//////////////轴位置赋初值////////////
IF arrAxisPar[AxisNo.BuffeLine].arrTargetPoint[1]=0 THEN
	arrAxisPar[AxisNo.BuffeLine].arrTargetPoint[1]:=20;
END_IF
IF arrAxisPar[AxisNo.Mould].arrTargetPoint[1]=0 THEN
	arrAxisPar[AxisNo.Mould].arrTargetPoint[1]:=230;
END_IF
IF arrAxisPar[AxisNo.Mould].arrTargetPoint[2]=0 THEN
	arrAxisPar[AxisNo.Mould].arrTargetPoint[2]:=130;
END_IF
IF arrAxisPar[AxisNo.Cuter].arrTargetPoint[1]=0 THEN
	arrAxisPar[AxisNo.Cuter].arrTargetPoint[1]:=230;
END_IF
IF arrAxisPar[AxisNo.Cuter].arrTargetPoint[2]=0 THEN
	arrAxisPar[AxisNo.Cuter].arrTargetPoint[2]:=130;
END_IF
IF arrAxisPar[AxisNo.CCDPressPush].arrTargetPoint[1]=0 THEN
	arrAxisPar[AxisNo.CCDPressPush].arrTargetPoint[1]:=200;
END_IF
IF arrAxisPar[AxisNo.CCDPressPush].arrTargetPoint[2]=0 THEN
	arrAxisPar[AxisNo.CCDPressPush].arrTargetPoint[2]:=180;
END_IF
(*
IF arrAxisPar[AxisNo.NGPush1].arrTargetPoint[1]=0 THEN
	arrAxisPar[AxisNo.NGPush1].arrTargetPoint[1]:=1;
END_IF
IF arrAxisPar[AxisNo.NGPush1].arrTargetPoint[2]=0 THEN
	arrAxisPar[AxisNo.NGPush1].arrTargetPoint[2]:=180;
END_IF
IF arrAxisPar[AxisNo.NGPush2].arrTargetPoint[1]=0 THEN
	arrAxisPar[AxisNo.NGPush2].arrTargetPoint[1]:=270;
END_IF
IF arrAxisPar[AxisNo.NGPush2].arrTargetPoint[2]=0 THEN
	arrAxisPar[AxisNo.NGPush2].arrTargetPoint[2]:=90;
END_IF
*)
IF arrAxisPar[AxisNo.MouldRectify_X].arrTargetPoint[1]=0 THEN
	arrAxisPar[AxisNo.MouldRectify_X].arrTargetPoint[1]:=1;
END_IF
IF arrAxisPar[AxisNo.MouldRectify_X].arrTargetPoint[2]=0 THEN
	arrAxisPar[AxisNo.MouldRectify_X].arrTargetPoint[2]:=2;
END_IF
IF arrAxisPar[AxisNo.MouldRectify_Y].arrTargetPoint[1]=0 THEN
	arrAxisPar[AxisNo.MouldRectify_Y].arrTargetPoint[1]:=1;
END_IF
IF arrAxisPar[AxisNo.MouldRectify_Y].arrTargetPoint[2]=0 THEN
	arrAxisPar[AxisNo.MouldRectify_Y].arrTargetPoint[2]:=2;
END_IF
IF arrAxisPar[AxisNo.CuterBeltChange].arrTargetPoint[1]=0 THEN
	arrAxisPar[AxisNo.CuterBeltChange].arrTargetPoint[1]:=1;
END_IF
IF arrAxisPar[AxisNo.CuterBeltChange].arrTargetPoint[2]=0 THEN
	arrAxisPar[AxisNo.CuterBeltChange].arrTargetPoint[2]:=2;
END_IF
IF arrAxisPar[AxisNo.CuterDegRectify].arrTargetPoint[1]=0 THEN
	arrAxisPar[AxisNo.CuterDegRectify].arrTargetPoint[1]:=0.1;
END_IF
IF arrAxisPar[AxisNo.CuterDegRectify].arrTargetPoint[2]=0 THEN
	arrAxisPar[AxisNo.CuterDegRectify].arrTargetPoint[2]:=0.2;
END_IF
//监控极耳数据
TabData[1].fPhotoPosC;TabData[1].fPhotoPosM;TabData[1].fTab_OffsetC;TabData[1].fTab_OffsetM;
TabData[2].fPhotoPosC;TabData[2].fPhotoPosM;TabData[2].fTab_OffsetC;TabData[2].fTab_OffsetM;
TabData[3].fPhotoPosC;TabData[3].fPhotoPosM;TabData[3].fTab_OffsetC;TabData[3].fTab_OffsetM;
TabData[4].fPhotoPosC;TabData[4].fPhotoPosM;TabData[3].fTab_OffsetC;TabData[4].fTab_OffsetM;
TabData[5].fPhotoPosC;TabData[5].fPhotoPosM;TabData[5].fTab_OffsetC;TabData[5].fTab_OffsetM;
TabData[6].fPhotoPosC;TabData[6].fPhotoPosM;TabData[6].fTab_OffsetC;TabData[6].fTab_OffsetM;
TabData[7].fPhotoPosC;TabData[7].fPhotoPosM;TabData[7].fTab_OffsetC;TabData[7].fTab_OffsetM;
TabData[8].fPhotoPosC;TabData[8].fPhotoPosM;TabData[8].fTab_OffsetC;TabData[8].fTab_OffsetM;
TabData[9].fPhotoPosC;TabData[9].fPhotoPosM;TabData[9].fTab_OffsetC;TabData[9].fTab_OffsetM;
TabData[10].fPhotoPosC;TabData[10].fPhotoPosM;TabData[10].fTab_OffsetC;TabData[10].fTab_OffsetM;
//监控极耳间距数据
InteData[1].fTabIntervalC;InteData[1].fTabIntervalM;InteData[1].bLineScanNG;
InteData[2].fTabIntervalC;InteData[2].fTabIntervalM;InteData[2].bLineScanNG;
InteData[3].fTabIntervalC;InteData[3].fTabIntervalM;InteData[3].bLineScanNG;
InteData[4].fTabIntervalC;InteData[4].fTabIntervalM;InteData[4].bLineScanNG;
InteData[5].fTabIntervalC;InteData[5].fTabIntervalM;InteData[5].bLineScanNG;
InteData[6].fTabIntervalC;InteData[6].fTabIntervalM;InteData[6].bLineScanNG;
InteData[7].fTabIntervalC;InteData[7].fTabIntervalM;InteData[7].bLineScanNG;
InteData[8].fTabIntervalC;InteData[8].fTabIntervalM;InteData[8].bLineScanNG;
InteData[9].fTabIntervalC;InteData[9].fTabIntervalM;InteData[9].bLineScanNG;
InteData[10].fTabIntervalC;InteData[10].fTabIntervalM;InteData[10].bLineScanNG;

IF bTest[1] THEN
	arrAxisCtrl[VirAxisNo.VirMain].Cmd.bDynamitcsParSel:=1;
	arrAxisCtrl[VirAxisNo.VirMain].Cmd.fPositon_of_Abs:=arrAxisCtrl[VirAxisNo.VirMain].Status.fActPos-arrAxisCtrl[VirAxisNo.VirMain].Status.fModuloActPos+720;
	//arrAxisPar[VirAxisNo.VirMain].fTagatTime:=((arrAxisCtrl[VirAxisNo.VirMain].Cmd.fPositon_of_Abs-arrAxisCtrl[VirAxisNo.VirMain].Status.fActPos)/360) *60/PolePar.iMainVel+0.05 ;
	arrAxisPar[VirAxisNo.VirMain].fVelocity_of_Abs:=PolePar.iMainVel*6;
	arrAxisCtrl[VirAxisNo.VirMain].Cmd.bMoveAbs:=TRUE;
	bTest[1]:=FALSE;
END_IF

ftest1:=FC_LengthToAngle(CCD_COM.fDemLength,PolePar.Machine.fMQDriverDiameter);
(*
arrAxisCtrl[VirAxisNo.VirMain].Status.Moving;     arrAxisCtrl[VirAxisNo.VirMain].Status.fActPos;
IF bTest[2] THEN
	arrAxisCtrl[VirAxisNo.VirMain].Cmd.bDynamitcsParSel:=1;
	ftest2:=arrAxisCtrl[VirAxisNo.VirMain].Status.fActPos+360;
	arrAxisCtrl[VirAxisNo.VirMain].Cmd.fPositon_of_Abs:=ftest2;
	//arrAxisPar[VirAxisNo.VirMain].fTagatTime:=((arrAxisCtrl[VirAxisNo.VirMain].Cmd.fPositon_of_Abs-arrAxisCtrl[VirAxisNo.VirMain].Status.fActPos)/360) *60/PolePar.iMainVel+0.05 ;
	arrAxisPar[VirAxisNo.VirMain].fVelocity_of_Abs:=20;
	arrAxisCtrl[VirAxisNo.VirMain].Cmd.bMoveAbs:=TRUE;
	itest:=2;
bTest[2]:=FALSE;
END_IF
IF bTest[3] THEN
	arrAxisCtrl[VirAxisNo.VirMain].Cmd.bDynamitcsParSel:=1;
	ftest3:=arrAxisCtrl[VirAxisNo.VirMain].Status.fActPos-arrAxisCtrl[VirAxisNo.VirMain].Status.fModuloActPos+720;
	arrAxisCtrl[VirAxisNo.VirMain].Cmd.fPositon_of_Abs:=ftest3;
	//arrAxisPar[VirAxisNo.VirMain].fTagatTime:=((arrAxisCtrl[VirAxisNo.VirMain].Cmd.fPositon_of_Abs-arrAxisCtrl[VirAxisNo.VirMain].Status.fActPos)/360) *60/PolePar.iMainVel+0.05 ;
	arrAxisPar[VirAxisNo.VirMain].fVelocity_of_Abs:=20;
	arrAxisCtrl[VirAxisNo.VirMain].Cmd.bMoveAbs:=TRUE;
	itest:=3;
bTest[3]:=FALSE;
END_IF
*)
IF btest[2] THEN
	MEMSET(ADR(fM_TabInterData),0,SIZEOF(fM_TabInterData)); //  
	btest[2]:=FALSE;
END_IF
IF btest[3] THEN
	MEMSET(ADR(fDriverOffsetData),0,SIZEOF(fDriverOffsetData)); //  
	btest[3]:=FALSE;
END_IF
IF btest[4] THEN
	//MEMSET(ADR(),0,SIZEOF()); //  
	btest[4]:=FALSE;
END_IF
IF btest[5] THEN
	//MEMSET(ADR(),0,SIZEOF()); //  
	btest[5]:=FALSE;
	fDegreeRec1:=FC_Variance(fOffsetDeg);		
END_IF



(*
IF NOT InterPart.M1Safety THEN
   arrAxisCtrl[AxisNo.SubBelt1].Cmd.JogP_Condition:=TRUE;
   arrAxisCtrl[AxisNo.SubBelt1].Cmd.JogN_Condition:=TRUE;
ELSE 
   arrAxisCtrl[AxisNo.SubBelt1].Cmd.JogP_Condition:=FALSE;
   arrAxisCtrl[AxisNo.SubBelt1].Cmd.JogN_Condition:=FALSE;
END_IF

IF NOT InterPart.M2Safety THEN
   arrAxisCtrl[AxisNo.SubBelt2].Cmd.JogP_Condition:=TRUE;
   arrAxisCtrl[AxisNo.SubBelt2].Cmd.JogN_Condition:=TRUE;
ELSE 
   arrAxisCtrl[AxisNo.SubBelt2].Cmd.JogP_Condition:=FALSE;
   arrAxisCtrl[AxisNo.SubBelt2].Cmd.JogN_Condition:=FALSE;
END_IF
 
IF NOT InterPart.M3Safety THEN
   arrAxisCtrl[AxisNo.SubBelt3].Cmd.JogP_Condition:=TRUE;
   arrAxisCtrl[AxisNo.SubBelt3].Cmd.JogN_Condition:=TRUE;
ELSE 
   arrAxisCtrl[AxisNo.SubBelt3].Cmd.JogP_Condition:=FALSE;
   arrAxisCtrl[AxisNo.SubBelt3].Cmd.JogN_Condition:=FALSE;
END_IF
*)



////位置参数固定
arrAxisPar[AxisNo.Mould].arrTargetPoint[1]:=270;
arrAxisPar[AxisNo.Mould].arrTargetPoint[2]:=120;
arrAxisPar[AxisNo.Cuter].arrTargetPoint[1]:=270;
arrAxisPar[AxisNo.Cuter].arrTargetPoint[2]:=70;

arrAxisPar[AxisNo.BuffeLine].arrTargetPoint[1]:=arrAxisPar[AxisNo.BuffeLine].arrTargetPoint[2]+61.5;
END_ACTION

ACTION F09INIT:
rtInit(CLK:=SysPart.hmiInit, Q=> );
tonInit[1](In:=,PT:=T#800MS);
tonInit[2](In:=,PT:=T#100MS);
CASE iInitstep OF
0:
	IF (SysPart.bInit AND NOT SysPart.bInitDone) OR rtInit.Q THEN
		SysPart.bInitDone:=FALSE;
		SysPart.bIniting:=TRUE;
		iInitstep:=10;
	END_IF
10://气缸类型初始化
//1:有磁性开关双控；2：有磁性开关单控；3：无磁性开关双控；4：无磁性开关单控；默认为1
	arrCyCtrl[CyNo.	Inflation_L	].Cmd.iType:=3;	(*左放卷气胀轴气缸*)	
	arrCyCtrl[CyNo.	Inflation_R	].Cmd.iType:=3;	(*右放卷气胀轴气缸*)	
	arrCyCtrl[CyNo.	BoardPressL	].Cmd.iType:=1;	(*左接带压板气缸*)	
	arrCyCtrl[CyNo.	BoardPressR	].Cmd.iType:=1;	(*右接带压板气缸*)	
	arrCyCtrl[CyNo.	DriverPressAux	].Cmd.iType:=1;	(*辅助驱动压辊气缸*)	
	arrCyCtrl[CyNo.	CoderRollPress	].Cmd.iType:=1;	(*编码器辊压辊气缸*)	
	arrCyCtrl[CyNo.	DriverPressDDR	].Cmd.iType:=1;	(*主驱动压辊气缸*)	
	arrCyCtrl[CyNo.	NGRevBeltUpDown	].Cmd.iType:=1;	(*踢废倒装皮带升降气缸*)	
	arrCyCtrl[CyNo.	NGRevBeltTension	].Cmd.iType:=3;	(*踢废倒装皮带张紧气缸*)	
	arrCyCtrl[CyNo.	PoleBrushDustPush_U	].Cmd.iType:=1;	(*极片上表面毛刷除尘升降缸*)	
	arrCyCtrl[CyNo.	PoleWindDustPush_U	].Cmd.iType:=1;	(*极片上表面风刀除尘升降缸*)	
	arrCyCtrl[CyNo.	PoleBrushDustPush_D	].Cmd.iType:=1;	(*极片下表面毛刷除尘升降缸*)	
	arrCyCtrl[CyNo.	PoleWindDustPush_D	].Cmd.iType:=1;	(*极片下表面风刀除尘升降缸*)	
	arrCyCtrl[CyNo.	DustRevBeltUpDown	].Cmd.iType:=1;	(*极片下表面除尘倒装皮带升降气缸*)	
	arrCyCtrl[CyNo.	NGBoxLock1	].Cmd.iType:=4;	(*NG料盒归正气缸1*)	
	arrCyCtrl[CyNo.	NGBoxLock2	].Cmd.iType:=4;	(*NG料盒归正气缸2*)	
	arrCyCtrl[CyNo.	WasteBoxPush	].Cmd.iType:=4;	(*连续废料收集箱推料气缸*)	
	
	arrCyCtrl[EvNo.	ConnectDustVacuo	].Cmd.iType:=4;	//	极片接带平台除尘真空	
	arrCyCtrl[EvNo.	LineSceneDustBlow	].Cmd.iType:=4;	//	线扫相机镜头除尘吹气	
	arrCyCtrl[EvNo.	LineSceneDustVacuo	].Cmd.iType:=4;	//	线扫相机镜头除尘真空	
	arrCyCtrl[EvNo.	AreaArrayDustBlow	].Cmd.iType:=4;	//	模切面阵相机镜头除尘吹气	
	arrCyCtrl[EvNo.	MouldUpBlow	].Cmd.iType:=3;	//	模具上模吹气	
	arrCyCtrl[EvNo.	MouldDownVacuo	].Cmd.iType:=4;	//	模具下模真空	
	arrCyCtrl[EvNo.	MouldDownAir	].Cmd.iType:=4;	//	模具下模破真空	
	arrCyCtrl[EvNo.	NGPushInsideAir	].Cmd.iType:=4;	//	NG踢废腔室破真空	
	arrCyCtrl[EvNo.	NGPushInsideVacuo	].Cmd.iType:=4;	//	NG踢废腔室真空	
	arrCyCtrl[EvNo.	BrushDustVacuo_U	].Cmd.iType:=4;	//	上表面毛刷除尘真空	
	arrCyCtrl[EvNo.	WindDustBlow_U	].Cmd.iType:=4;	//	上表面风刀除尘吹气	
	arrCyCtrl[EvNo.	WindDustVacuo_U	].Cmd.iType:=4;	//	上表面风刀除尘真空	
	arrCyCtrl[EvNo.	BrushDustVacuo_D	].Cmd.iType:=4;	//	下表面毛刷除尘真空	
	arrCyCtrl[EvNo.	WindDustBlow_D	].Cmd.iType:=4;	//	下表面风刀除尘吹气	
	arrCyCtrl[EvNo.	WindDustVacuo_D	].Cmd.iType:=4;	//	下表面风刀除尘真空	
	arrCyCtrl[EvNo.	RJ_Blow	].Cmd.iType:=4;	//	下表面风刀除尘真空		
	arrCyCtrl[EvNo.	RJDustBlow  ].Cmd.iType:=4;	//R角风刀吹气	
	
	iInitstep:=20;

20://判断是否在耦合中
	IF arrAxis[AxisNo.BuffeLine].Status.Coupled THEN
		arrAxisCtrl[AxisNo.BuffeLine].Cmd.bStop:=TRUE;
	END_IF
	IF arrAxis[AxisNo.DriverDDR].Status.Coupled THEN
		arrAxisCtrl[AxisNo.DriverDDR].Cmd.bStop:=TRUE;
	END_IF	
	IF arrAxis[AxisNo.Mould].Status.Coupled THEN
		arrAxisCtrl[AxisNo.Mould].Cmd.bStop:=TRUE;
	END_IF		
	IF arrAxis[AxisNo.Cuter].Status.Coupled THEN
		arrAxisCtrl[AxisNo.Cuter].Cmd.bStop:=TRUE;
	END_IF		
	IF arrAxis[AxisNo.CCDPressPush].Status.Coupled THEN
		arrAxisCtrl[AxisNo.CCDPressPush].Cmd.bStop:=TRUE;
	END_IF	
	IF arrAxis[VirAxisNo.VirBelt].Status.Coupled THEN
		arrAxisCtrl[VirAxisNo.VirBelt].Cmd.bStop:=TRUE;
	END_IF	
	(*
	IF arrAxis[AxisNo.NGPush2].Status.Coupled THEN
		arrAxisCtrl[AxisNo.NGPush2].Cmd.bStop:=TRUE;
	END_IF	
	*)
	IF NOT arrAxis[AxisNo.BuffeLine].Status.Coupled AND NOT arrAxis[AxisNo.DriverDDR].Status.Coupled AND NOT arrAxis[AxisNo.Mould].Status.Coupled AND
		NOT arrAxis[AxisNo.Cuter].Status.Coupled AND NOT arrAxis[AxisNo.CCDPressPush].Status.Coupled AND NOT arrAxis[VirAxisNo.VirBelt].Status.Coupled(* AND
		NOT arrAxis[AxisNo.NGPush2].Status.Coupled *)THEN
		iInitstep:=30;
	END_IF
	
30://凸轮创建信号复位
	stPoleBufferCam.bCreatTable:=FALSE;
	stVirBeltCam.bCreatTable:=FALSE;
	//stNGPushCam.bCreatTable:=FALSE;
	stCuterCam.bCreatTable:=FALSE;
	stDriverCam.bCreatTable:=FALSE;
	stMouldCam.bCreatTable:=FALSE;
	stCCDPressCam.bCreatTable:=FALSE;
	stPoleBufferCam_1.bCreatTable:=FALSE;
	stVirDriverCam.bCreatTable:=FALSE;
	
	FOR i:=1 TO 50 DO//NG类型标志位复位
		Production.NGFlag[i]:=FALSE;
	END_FOR
	iInitstep:=40;
	
40://凸轮创建
	stVirBeltCam.bCreatTable:=TRUE;
	//stNGPushCam.bCreatTable:=TRUE;
	stCuterCam.bCreatTable:=TRUE;
	stDriverCam.bCreatTable:=TRUE;
	stMouldCam.bCreatTable:=TRUE;
	stCCDPressCam.bCreatTable:=TRUE;
	stVirDriverCam.bCreatTable:=TRUE;
	iInitstep:=50;
	
50://凸轮创建判断
IF NOT tonInit[2].Q THEN
	tonInit[2].IN:=TRUE;
ELSE
	IF stVirBeltCam.bCreatTableDone (*AND stNGPushCam.bCreatTableDone*) AND
		stCuterCam.bCreatTableDone AND stDriverCam.bCreatTableDone AND stMouldCam.bCreatTableDone AND
		stCCDPressCam.bCreatTableDone AND stVirDriverCam.bCreatTableDone THEN
		stVirBeltCam.bCreatTable:=FALSE;
		//stNGPushCam.bCreatTable:=FALSE;
		stCuterCam.bCreatTable:=FALSE;
		stDriverCam.bCreatTable:=FALSE;
		stMouldCam.bCreatTable:=FALSE;
		stCCDPressCam.bCreatTable:=FALSE;	
		stVirDriverCam.bCreatTable:=FALSE;
		tonInit[2].IN:=FALSE;	
		iInitstep:=60;
	END_IF
END_IF

60://极片缓存凸轮创建
	stPoleBufferCam.bCreatTable:=TRUE;
	stPoleBufferCam_1.bCreatTable:=TRUE;
	iInitstep:=70;
	
70://判断极片缓存凸轮创建	
	IF stPoleBufferCam.bCreatTableDone AND stPoleBufferCam_1.bCreatTableDone THEN
		stPoleBufferCam.bCreatTable:=FALSE;	
		stPoleBufferCam_1.bCreatTable:=FALSE;	
		iInitstep:=80;
	END_IF

80://完成
	SysPart.bInit:=FALSE;
	IF stSysState.iMode=0 THEN
		SysPart.bInitDone:=TRUE;
		SysPart.bIniting:=FALSE;
		iInitstep:=0;
	ELSE
		IF NOT tonInit[1].Q THEN
			tonInit[1].IN:=TRUE;
		ELSE
			SysPart.hmiInit:=FALSE;
			SysPart.bIniting:=FALSE;
			SysPart.bInitDone:=TRUE;
			tonInit[1].IN:=FALSE;
			iInitstep:=0;	
		END_IF	
	END_IF
END_CASE
END_ACTION

ACTION F10GearCall:
(*
//虚拟放卷
fbVirDriverGear(
	Reset:=stSysState.bReset , 
	fratio1:= , 
	bError=>stVirDriverGear.bError , 
	bReady=>stVirDriverGear.bReady , 
	InGear=>stVirDriverGear.bInGear , 
	bEnable:=stVirDriverGear.bEnable , 
	bGearOutMode:=stVirDriverGear.bGearOutMode , 
	master:=arrAxis[VirAxisNo.VirMain] , 
	slave1:=arrAxis[VirAxisNo.VirDriver] );
*)
fbVDriverCam(
	Reset:=stSysState.bReset , 
	bCamInExecute:=FALSE , //stVirDriverCam.bCamInExecute
	bCreatTable:=stVirDriverCam.bCreatTable , 
	iTable:=TableNo.VirDirver , 
	fCompensation:= , //主驱运动时片宽的补偿值
	fDiameterDriver:=PolePar.Machine.fMQDriverDiameter , 
	fPoleWidth:=PolePar.fPoleWidth , 
	fMainPos:=ProductPar.parPublic.fMainPos , 
	
	axisSlave:=arrAxis[VirAxisNo.VirDriver]   , 
	axisMaster:= arrAxis[VirAxisNo.VirMain], 
	
	bCreatTableDone=>stVirDriverCam.bCreatTableDone , 
	bCreatTableError=>stVirDriverCam.bCreatTableError , 
	bError=>stVirDriverCam.bError , 
	bReady=>stVirDriverCam.bReady , 
	bInSync=>stVirDriverCam.bInSync );	


	

	
	
//裁切输送皮带	
fbCuterBeltGear(	
	Reset:=stSysState.bReset , 
	fratio1:=PolePar.Machine.fBelt5Scaling   ,  //PolePar.Machine.fBelt1Scaling
	bError=>stCuterBeltGear.bError , 
	bReady=>stCuterBeltGear.bReady , 
	InGear=>stCuterBeltGear.bInGear , 
	bEnable:=stCuterBeltGear.bEnable , 
	bGearOutMode:=stCuterBeltGear.bGearOutMode , 
	master:=arrAxis[VirAxisNo.VirBelt] , 
	slave1:=arrAxis[AxisNo.CuterBelt] );
	PolePar.Machine.fBelt1Scaling:=1;
//踢废倒装皮带	
fbNGReverseBeltGear(	
	Reset:=stSysState.bReset , 
	fratio1:=PolePar.Machine.fBelt5Scaling , 
	bError=>stNGReverseBeltGear.bError , 
	bReady=>stNGReverseBeltGear.bReady , 
	InGear=>stNGReverseBeltGear.bInGear , 
	bEnable:=stNGReverseBeltGear.bEnable , 
	bGearOutMode:=stNGReverseBeltGear.bGearOutMode , 
	master:=arrAxis[VirAxisNo.VirBelt] , 
	slave1:=arrAxis[AxisNo.NGPushReverseBelt] );
	PolePar.Machine.fBelt2Scaling:=1;
//上表面除尘皮带	
fbDedustBeltGear(	
	Reset:=stSysState.bReset , 
	fratio1:=PolePar.Machine.fBelt5Scaling , 
	bError=>stDedustBeltGear.bError , 
	bReady=>stDedustBeltGear.bReady , 
	InGear=>stDedustBeltGear.bInGear , 
	bEnable:=stDedustBeltGear.bEnable , 
	bGearOutMode:=stDedustBeltGear.bGearOutMode , 
	master:=arrAxis[VirAxisNo.VirBelt] , 
	slave1:=arrAxis[AxisNo.DedustBelt] );
	PolePar.Machine.fBelt3Scaling:=1;
//下表面除尘倒装皮带	
fbDedustReverseBeltGear(	
	Reset:=stSysState.bReset , 
	fratio1:=PolePar.Machine.fBelt5Scaling , 
	bError=>stDedustReverseBeltGear.bError , 
	bReady=>stDedustReverseBeltGear.bReady , 
	InGear=>stDedustReverseBeltGear.bInGear , 
	bEnable:=stDedustReverseBeltGear.bEnable , 
	bGearOutMode:=stDedustReverseBeltGear.bGearOutMode , 
	master:=arrAxis[VirAxisNo.VirBelt] , 
	slave1:=arrAxis[AxisNo.DedustReverseBelt] );
	PolePar.Machine.fBelt4Scaling:=1;
	arrAxisCtrl[AxisNo.DedustReverseBelt].Status.Moving;
//分段主皮带1	
bSubBelt1fratio:=TRUE;//屏蔽1号皮带时，置false
IF bSubBelt1fratio THEN
	fbSubBelt1Gear.fratio1:=PolePar.Machine.fBelt5Scaling;
ELSE
	fbSubBelt1Gear.fratio1:=0;
END_IF
fbSubBelt1Gear(	
	Reset:=stSysState.bReset , 
	fratio1:= , 
	bError=>stSubBelt1Gear.bError , 
	bReady=>stSubBelt1Gear.bReady , 
	InGear=>stSubBelt1Gear.bInGear , 
	bEnable:=stSubBelt1Gear.bEnable , 
	bGearOutMode:=stSubBelt1Gear.bGearOutMode , 
	master:=arrAxis[VirAxisNo.VirBelt] , 
	slave1:=arrAxis[AxisNo.SubBelt1] );
	
//分段主皮带2	
IF bSubBelt2fratio THEN
	fbSubBelt2Gear.fratio1:=PolePar.Machine.fBelt6Scaling;
ELSE
	fbSubBelt2Gear.fratio1:=0;
END_IF
fbSubBelt2Gear(	
	Reset:=stSysState.bReset , 
	fratio1:= , 
	bError=>stSubBelt2Gear.bError , 
	bReady=>stSubBelt2Gear.bReady , 
	InGear=>stSubBelt2Gear.bInGear , 
	bEnable:=stSubBelt2Gear.bEnable , 
	bGearOutMode:=stSubBelt2Gear.bGearOutMode , 
	master:=arrAxis[VirAxisNo.VirBelt] , 
	slave1:=arrAxis[AxisNo.SubBelt2] );
	
//分段主皮带3	
IF bSubBelt3fratio THEN
	fbSubBelt3Gear.fratio1:=PolePar.Machine.fBelt7Scaling;
ELSE
	fbSubBelt3Gear.fratio1:=0;
END_IF
fbSubBelt3Gear(	
	Reset:=stSysState.bReset , 
	fratio1:= , 
	bError=>stSubBelt3Gear.bError , 
	bReady=>stSubBelt3Gear.bReady , 
	InGear=>stSubBelt3Gear.bInGear , 
	bEnable:=stSubBelt3Gear.bEnable , 
	bGearOutMode:=stSubBelt3Gear.bGearOutMode , 
	master:=arrAxis[VirAxisNo.VirBelt] , 
	slave1:=arrAxis[AxisNo.SubBelt3] );
END_ACTION

ACTION F11CamCall:
//极片缓存 V1

fbPoleBufferCam(
	Reset:=stSysState.bReset , 
	bCamInExecute:=FALSE , //stPoleBufferCam.bCamInExecute
	bCreatTable:=stPoleBufferCam.bCreatTable , 
	iTable:=TableNo.BufferLine , 
	iTableMQDriver:=TableNo.Dirver , 
	iTableVirDriver:=TableNo.VirDirver , 
	fDiameterDriver:=PolePar.Machine.fMQDriverDiameter , 
	fCompensation:=fPoleBufferCompensation , 
	fPoleWidth:=PolePar.fPoleWidth , 
	fDriverEndPosInCam:=ProductPar.parPublic.fMainPos , 
	axisSlave:=arrAxis[AxisNo.BuffeLine] , 
	axisMaster:=arrAxis[VirAxisNo.VirMain] , 
	bCreatTableDone=>stPoleBufferCam.bCreatTableDone , 
	bCreatTableError=>stPoleBufferCam.bCreatTableError , 
	bError=>stPoleBufferCam.bError , 
	bReady=>stPoleBufferCam.bReady , 
	bInSync=>stPoleBufferCam.bInSync );
	
fbPoleBufferCam_1(
	Reset:=stSysState.bReset , 
	bCamInExecute:=FALSE , //stPoleBufferCam_1.bCamInExecute 
	bCreatTable:=stPoleBufferCam_1.bCreatTable , 
	iTable:=TableNo.BufferLine_1 , 
	iTableMQDriver:=TableNo.Dirver , 
	iTableVirDriver:=TableNo.VirDirver , 
	fDiameterDriver:=PolePar.Machine.fMQDriverDiameter , 
	fCompensation:=fPoleBufferCompensation , 
	fPoleWidth:=PolePar.fPoleWidth , 
	fDriverEndPosInCam:=ProductPar.parPublic.fMainPos , 
	axisSlave:=arrAxis[AxisNo.BuffeLine] , 
	axisMaster:=arrAxis[VirAxisNo.VirMain] , 
	bCreatTableDone=>stPoleBufferCam_1.bCreatTableDone , 
	bCreatTableError=>stPoleBufferCam_1.bCreatTableError , 
	bError=>stPoleBufferCam_1.bError , 
	bReady=>stPoleBufferCam_1.bReady , 
	bInSync=>stPoleBufferCam_1.bInSync );

	
	
	
(*
//极片缓存 V2
fbPoleBufferCam(
	Reset:=stSysState.bReset , 
	bCamInExecute:=stPoleBufferCam.bCamInExecute , 
	bCreatTable:=stPoleBufferCam.bCreatTable , 
	iTable:=TableNo.BufferLine , 
	iTableMQDriver:=TableNo.Dirver , 
	fDiameterDriver:=PolePar.Machine.fMQDriverDiameter , 
	fCompensation:= , 
	fPoleWidth:=PolePar.fPoleWidth , 
	fDriverEndPosInCam:=ProductPar.parPublic.fMainPos , 
	axisSlave:=arrAxis[AxisNo.BuffeLine] , 
	axisMaster:=arrAxis[VirAxisNo.VirMain] , 
	bCreatTableDone=>stPoleBufferCam.bCreatTableDone , 
	bCreatTableError=>stPoleBufferCam.bCreatTableError , 
	bError=>stPoleBufferCam.bError , 
	bReady=>stPoleBufferCam.bReady , 
	bInSync=>stPoleBufferCam.bInSync );
*)
(*
fbAuxDriverTen2.fratio1    :=PolePar.Machine.fMQDriverDiameter*pi/720;
fbAuxDriverTen2.fratio2    :=-PolePar.Machine.fAuxDriverInDiameter*pi/720;
fbAuxDriverTen2(
	Reset:= stSysState.bReset, 
	fratio1:= , 
	fratio2:= , 
	bError=> , 
	bReady=> , 
	InGear=> , 
	bEnable:=       bEnable , 
	master1:=       arrAxis[AxisNo.DriverDDR] , 
	master2:=       arrAxis[AxisNo.DriverAux], 
	slave1:=          arrAxis[AxisNo.BuffeLine]);
fbAuxDriverTen2.bReady;
fbAuxDriverTen2.InGear;
fbAuxDriverTen2.InGear;


fbTensionVirDriver(
	bReset:=                stSysState.bReset,  
    bTenExecute:=        bEnable2 , 
	PidSwitch:=                                     , 
	fActBufferPos:=     arrAxis[AxisNo.BuffeLine].NcToPlc.ActPos, 

	fBufferrMinPos:=    PolePar.MQ.BufferMinPos,   
	fBufferMaxPos:=     PolePar.MQ.BufferMaxPos, 
	fBufferBlancePos:=  PolePar.MQ.BufferBlancePos , 

	fWith:=                               , 
	bReady=>                          , 
	bTensionOK=>                   , 
	bError=>                           , 

    virMain:=            arrAxis[VirAxisNo.VirMain] , 
	TimerAxis:=         arrAxis[AxisNo.DriverDDR] , 
   	Slave:=                arrAxis[VirAxisNo.VirDriver]  );

fbTensionVirDriver.bReady;
fbTensionVirDriver.bTensionOK;
fbTensionVirDriver.bError;
*)















//主驱动
fbDriverCam(
	Reset:=stSysState.bReset , 
	bCamInExecute:=stDriverCam.bCamInExecute , 
	bCreatTable:=stDriverCam.bCreatTable , 
	iTable:=TableNo.Dirver , 
	fCompensation:= , //主驱运动时片宽的补偿值
	fDiameterDriver:=PolePar.Machine.fMQDriverDiameter , 
	fPoleWidth:=PolePar.fPoleWidth , 
	fMainPos:=ProductPar.parPublic.fMainPos , 
	axisSlave:=arrAxis[AxisNo.DriverDDR]  , 
	axisMaster:= arrAxis[VirAxisNo.VirMain], 
	bCreatTableDone=>stDriverCam.bCreatTableDone , 
	bCreatTableError=>stDriverCam.bCreatTableError , 
	bError=>stDriverCam.bError , 
	bReady=>stDriverCam.bReady , 
	bInSync=>stDriverCam.bInSync );

//模具切刀
fbMouldCam(
	Reset:=stSysState.bReset , 
	bCamInExecute:=stMouldCam.bCamInExecute , 
	bCreatTable:=stMouldCam.bCreatTable , 
	iTable:=TableNo.Mould , 
	iTableSel:= , 
	fEnterPos:=arrAxisPar[AxisNo.Mould].arrTargetPoint[2] , 
	fLeavePos:=arrAxisPar[AxisNo.Mould].arrTargetPoint[1] , 
	fMainPos:=ProductPar.parPublic.fMainPos , 
	axisSlave:=arrAxis[AxisNo.Mould] , 
	axisMaster:=arrAxis[VirAxisNo.VirMain] , 
	bCreatTableDone=>stMouldCam.bCreatTableDone , 
	bCreatTableError=>stMouldCam.bCreatTableError , 
	bError=>stMouldCam.bError , 
	bReady=>stMouldCam.bReady , 
	bInSync=>stMouldCam.bInSync );
	
//裁切切刀
fbCuterCam(
	Reset:=stSysState.bReset , 
	bCamInExecute:=stCuterCam.bCamInExecute , 
	bCreatTable:=stCuterCam.bCreatTable , 
	iTable:=TableNo.Cuter , 
	iTableSel:= ,
	fEnterPos:=arrAxisPar[AxisNo.Cuter].arrTargetPoint[2] , //裁切切入点角度
	fLeavePos:=arrAxisPar[AxisNo.Cuter].arrTargetPoint[1] , //裁切切尽点角度
	fMainPos:=ProductPar.parPublic.fMainPos , 
	axisSlave:=arrAxis[AxisNo.Cuter] , 
	axisMaster:=arrAxis[VirAxisNo.VirMain] , 
	bCreatTableDone=>stCuterCam.bCreatTableDone , 
	bCreatTableError=>stCuterCam.bCreatTableError , 
	bError=>stCuterCam.bError , 
	bReady=>stCuterCam.bReady , 
	bInSync=>stCuterCam.bInSync );

//CCD压片升降
fbCCDPressCam(
	Reset:=stSysState.bReset , 
	bCamInExecute:=stCCDPressCam.bCamInExecute , 
	bCreatTable:=stCCDPressCam.bCreatTable , 
	iTable:=TableNo.CCDPress , 
	fMainPos:=ProductPar.parPublic.fMainPos , 
	fPressPos:=arrAxisPar[AxisNo.CCDPressPush].arrTargetPoint[2]  , 
	fLeavePos:=arrAxisPar[AxisNo.CCDPressPush].arrTargetPoint[1] , 
	axisSlave:=arrAxis[AxisNo.CCDPressPush]  , 
	axisMaster:=arrAxis[VirAxisNo.VirMain]  , 
	bCreatTableDone=>stCCDPressCam.bCreatTableDone , 
	bCreatTableError=>stCCDPressCam.bCreatTableError , 
	bError=>stCCDPressCam.bError , 
	bReady=>stCCDPressCam.bReady , 
	bInSync=>stCCDPressCam.bInSync );
	
//皮带虚轴
fbVirBeltCam(
	Reset:=stSysState.bReset , 
	bCamInExecute:=stVirBeltCam.bCamInExecute , 
	bCreatTable:=stVirBeltCam.bCreatTable , 
	iTable:=TableNo.VirBelt , 
	fMainPos:=ProductPar.parPublic.fMainPos , 
	fBeltSpacePos:=PolePar.fBeltSpacePos , 
	axisSlave:=arrAxis[VirAxisNo.VirBelt]  , 
	axisMaster:=arrAxis[VirAxisNo.VirMain] , 
	bCreatTableDone=>stVirBeltCam.bCreatTableDone , 
	bCreatTableError=>stVirBeltCam.bCreatTableError , 
	bError=>stVirBeltCam.bError , 
	bReady=>stVirBeltCam.bReady , 
	bInSync=>stVirBeltCam.bInSync );
(*	
//NG踢料
fbNGPushCam(
	Reset:=stSysState.bReset , 
	bCamInExecute:=stNGPushCam.bCamInExecute , 
	bCreatTable:=stNGPushCam.bCreatTable , 
	iTable:=TableNo.NgPush , 
	iTableSel:= , 
	fEnterPos:=arrAxisPar[AxisNo.NGPush2].arrTargetPoint[2] , //NG打料预踢角度 , 
	fLeavePos:=arrAxisPar[AxisNo.NGPush2].arrTargetPoint[1] , //NG打料踢后角度 , 
	fMainPos:=ProductPar.parPublic.fMainPos , 
	axisSlave:=arrAxis[AxisNo.NGPush2] , 
	axisMaster:=arrAxis[VirAxisNo.VirMain] , 
	bCreatTableDone=>stNGPushCam.bCreatTableDone , 
	bCreatTableError=>stNGPushCam.bCreatTableError , 
	bError=>stNGPushCam.bError , 
	bReady=>stNGPushCam.bReady , 
	bInSync=>stNGPushCam.bInSync );
	*)
END_ACTION

ACTION F12TensionCall:


	fbPoleBufferTen.bTensionOK:=stUwindTen.bTensionOK;
	
	fbPoleBufferTen(
	bReset:=                               stSysState.bReset , 
	fAuxDriverDiameter:=            PolePar.Machine.fAuxDriverInDiameter ,  
	fDDRDiameter:=                    PolePar.Machine.fMQDriverDiameter ,  
	fPoleWith:=                           PolePar.fPoleWidth , 
    fCompensation:=                   fPoleBufferCompensation , 
    fDanceBlancePos:=                arrAxisPar[AxisNo.BuffeLine].arrTargetPoint[1] ,  
   	bPositiveLimit:=                     arrAxisCtrl[AxisNo.BuffeLine].Io.biPosLimit   , 
	bNegativeLimit:=                   arrAxisCtrl[AxisNo.BuffeLine].Io.biNegLimit      , 
	bTensionOK:=                       fbPoleBufferTen.bTensionOK     , 
	fMainVel:=                            PolePar.iMainVel         , 
	bReady=>                            stBufferTen.bReady , 
	bError=>                              stBufferTen.bError , 
	bInSync=>                            stBufferTen.bInSync, 
	VirMain:=                             arrAxis[VirAxisNo.VirMain], 
	//AuxDriver:=                          arrAxis[AxisNo.DriverAux] ,
	DDRDriver:=                         arrAxis[AxisNo.DriverDDR]  ,
	VirDriver:=                           arrAxis[VirAxisNo.VirDriver]  ,
	BufferLine:=                         arrAxis[AxisNo.BuffeLine] ,  
	bTenExecute:=                     stBufferTen.bExecute   );
	
	//放卷张力
PolePar.MQ.TenCcw_WindL:=PolePar.MQ.TenCcw_WindR:=FALSE;
	fbUwindTen(
		bReset:=stSysState.bReset , 
		bCcwL:=PolePar.MQ.TenCcw_WindL, //左放卷方向
		bCcwR:=PolePar.MQ.TenCcw_WindR,//右放卷方向
		bWindSel:=PolePar.MQ.bWindSelect, //左右卷选择
		fDiaMin:=250,//最小卷径		
		fDiaMax:=800,//最大卷径
		//fDanserDegree:=arrAxisCtrl[AxisNo.PoleTension].Status.fActPos , 
		fActTorque:= SEL(iPartSelect=1   , iActDriveTorque[2],    iActDriveTorque[1] )    , 
		fSetTorque:= SEL(iPartSelect=1   , iTargetTorque[2],       iTargetTorque[1] )      , 
		PidSwitch:=PolePar.MQ.WindPidSwitch ,
		bTenExecute:=stUwindTen.bTenExecute , 
		bStudyExecute:=stUwindTen.bStudyExecute AND stUwindTen.fStudyDiameter>0, 
		fStudyDiameter:=stUwindTen.fStudyDiameter , 
		fDriveDiameter:=PolePar.Machine.fMQDriverDiameter, 
		fPoleWith:=PolePar.fPoleWidth , 
		fCompensation:= , 
		fDancerMinPos:=PolePar.MQ.AuxDriverTenMinPos,//摆杆最小角度
		fDancerMaxPos:=PolePar.MQ.AuxDriverTenMaxPos,//摆杆最大角度
		fDanceBlancePos:=PolePar.MQ.AuxDriverTenBlancePos , //摆杆平衡角度
		fDanserDegree:=stAuxDriverTen.fDanserDegree , //摆杆实时角度
		//fDancerMinPos:=PolePar.MQ.WindTenMinPos , 
		//fDancerMaxPos:=PolePar.MQ.WindTenMaxPos , 
		//fDanceBlancePos:=PolePar.MQ.WindTenBlancePos , 
		bReady=>stUwindTen.bReady , 
		bTensionOK=>stUwindTen.bTensionOK , 
		bError=>stUwindTen.bError , 
		fWindDiameterTemp=>stUwindTen.fWindDiameter,
		VirMain:=arrAxis[VirAxisNo.VirMain] , 
		Master:=arrAxis[VirAxisNo.VirDriver] , 
		SlaveL:=arrAxis[AxisNo.UnWind_L], 
		SlaveR:=arrAxis[AxisNo.UnWind_R], 
		Driver:=arrAxis[AxisNo.DriverDDR] , 
		TimerAxis:=arrAxis[NameNo.VirTimeWind] , 
		TensionAxis:=arrAxis[AxisNo.PoleTension] , 
		Table:=PolePar.MQ.WindTenTable ,
		AxisNoBuffeLine :=AxisNo.BuffeLine);
	

		
		
(*
//左放卷张力

fbUwindLTen(
	bReset:=stSysState.bReset , 
	bCcw:=PolePar.MQ.TenCcw_WindL , 
	fDanserDegree:=stUwindLTen.fDanserDegree , 
	//fWindDiameter:=stUwindLTen.fWindDiameter  , 
	fActTorque:= SEL(iPartSelect=1   , iActDriveTorque[2],    iActDriveTorque[1] )    , 
	fSetTorque:= SEL(iPartSelect=1   , iTargetTorque[2],       iTargetTorque[1] )      , 
	PidSwitch:=TRUE , //PolePar.MQ.WindPidSwitch
	bTenExecute:=stUwindLTen.bTenExecute , 
	bStudyExecute:=stUwindLTen.bStudyExecute , 
	fStudyDiameter:=stUwindLTen.fStudyDiameter , 
	fDriveDiameter:=PolePar.Machine.fAuxDriverInDiameter , 
	fPoleWith:=PolePar.fPoleWidth , 
	fCompensation:= , 
	fDancerMinPos:=PolePar.MQ.WindTenMinPos , 
	fDancerMaxPos:=PolePar.MQ.WindTenMaxPos , 
	fDanceBlancePos:=PolePar.MQ.WindTenBlancePos , 
	bReady=>stUwindLTen.bReady , 
	bTensionOK=>stUwindLTen.bTensionOK , 
	bError=>stUwindLTen.bError , 
	VirMain:=arrAxis[VirAxisNo.VirMain] , 
	Master:=arrAxis[VirAxisNo.VirDriver] , 
	Slave:=arrAxis[AxisNo.UnWind_L] , 
	Driver:=arrAxis[AxisNo.DriverAux] , 
	TimerAxis:=arrAxis[NameNo.VirTimeWind] , 
	TensionAxis:=arrAxis[AxisNo.PoleTension] , 
	Table:=PolePar.MQ.WindTenTable );
	stUwindLTen.fDanserDegree:=arrAxisCtrl[AxisNo.PoleTension].Status.fActPos;
	PolePar.MQ.TenCcw_WindL:=FALSE;
	
	stUwindLTen.fWindDiameter  ;
	fbUwindLTen.fWindDiameter;
	fbUwindLTen.fDiameterCalculate;
	fbUwindLTen.fWindDiameterTemp;
	
//右放卷张力
fbUwindRTen(	
	bReset:=stSysState.bReset , 
	bCcw:=PolePar.MQ.TenCcw_WindR , 
	fDanserDegree:=stUwindRTen.fDanserDegree , 
	//fWindDiameter:=stUwindRTen.fWindDiameter , 
	fActTorque:= SEL(iPartSelect=1   , iActDriveTorque[2],    iActDriveTorque[1] )    , 
	fSetTorque:= SEL(iPartSelect=1   , iTargetTorque[2],       iTargetTorque[1] )      , 
	PidSwitch:=TRUE, //PolePar.MQ.WindPidSwitch 
	bTenExecute:=stUwindRTen.bTenExecute , 
	bStudyExecute:=stUwindRTen.bStudyExecute , 
	fStudyDiameter:=stUwindRTen.fStudyDiameter , 
	fDriveDiameter:=PolePar.Machine.fAuxDriverInDiameter , 
	fPoleWith:=PolePar.fPoleWidth , 
	fCompensation:= ,
	fDancerMinPos:=PolePar.MQ.WindTenMinPos , 
	fDancerMaxPos:=PolePar.MQ.WindTenMaxPos , 
	fDanceBlancePos:=PolePar.MQ.WindTenBlancePos , 
	bReady=>stUwindRTen.bReady , 
	bTensionOK=>stUwindRTen.bTensionOK , 
	bError=>stUwindRTen.bError , 
	VirMain:=arrAxis[VirAxisNo.VirMain] , 
	Master:=arrAxis[VirAxisNo.VirDriver] , 
	Slave:=arrAxis[AxisNo.UnWind_R]  , 
	Driver:=arrAxis[AxisNo.DriverAux] , 
	TimerAxis:=arrAxis[NameNo.VirTimeWind], 
	TensionAxis:=arrAxis[AxisNo.PoleTension] , 
	Table:=PolePar.MQ.WindTenTable );
	
	
	
	stUwindRTen.fDanserDegree:=arrAxisCtrl[AxisNo.PoleTension].Status.fActPos;
	PolePar.MQ.TenCcw_WindR:=FALSE;
	
	stUwindRTen.fWindDiameter  ;
	fbUwindRTen.fWindDiameter;
	fbUwindRTen.fDiameterCalculate;
	fbUwindRTen.fWindDiameterTemp;
*)	
//辅驱张力
stAuxDriverTen.fWindDiameter:=stAuxDriverTen.fStudyDiameter:=PolePar.Machine.fAuxDriverInDiameter;
PolePar.MQ.TenCcw_AuxDriver:=FALSE;
fbAuxDriverTen(
	bReset:=stSysState.bReset , 
	bCcw:=PolePar.MQ.TenCcw_AuxDriver , 
	fDanserDegree:=stAuxDriverTen.fDanserDegree , 
	fWindDiameter:=stAuxDriverTen.fWindDiameter , 
	PidSwitch:=FALSE , //PolePar.MQ.AuxDriverPidSwitch
	bTenExecute:=stAuxDriverTen.bTenExecute , 
	bStudyExecute:=FALSE, //stAuxDriverTen.bStudyExecute
	fStudyDiameter:=stAuxDriverTen.fStudyDiameter , 
	fPoleWith:=PolePar.fPoleWidth , 
	fCompensation:= , 
	fDancerMinPos:=PolePar.MQ.AuxDriverTenMinPos , 
	fDancerMaxPos:=PolePar.MQ.AuxDriverTenMaxPos , 
	fDanceBlancePos:=PolePar.MQ.AuxDriverTenBlancePos , 
	bReady=>stAuxDriverTen.bReady , 
	bTensionOK=>stAuxDriverTen.bTensionOK , 
	bError=>stAuxDriverTen.bError , 
	VirMain:=arrAxis[VirAxisNo.VirMain] , 
	Master:=arrAxis[VirAxisNo.VirDriver] , 
	Slave:=arrAxis[AxisNo.DriverAux] , 
	TimerAxis:=arrAxis[NameNo.VirTimeWind] , 
	Table:=PolePar.MQ.AuxDriverTenTable );
END_ACTION

ACTION F13ClearBelt:
//一键皮带清料
rtClearBelt[1](CLK:=SysPart.hmiClearBelt , Q=> );
rtClearBelt[2](CLK:= , Q=> );
rtClearBelt[3](CLK:= , Q=> );
rtClearBelt[4](CLK:= , Q=> );
rtClearBelt[5](CLK:= , Q=> );
tonClearBelt[1](In:=,PT:=T#200MS);
tonClearBelt[2](In:=,PT:=T#200MS);
tonClearBelt[3](In:=,PT:=T#200MS);
tonClearBelt[4](In:=,PT:=T#200MS);	
tonClearBelt[5](In:=,PT:=T#200MS);	
tonClearBelt[6](In:=,PT:=T#200MS);	
tonClearBelt[7](In:=,PT:=T#200MS);
tonClearBelt[8](In:=,PT:=T#200MS);
tonClearBelt[9](In:=,PT:=T#200MS);
tonClearBelt[10](In:=,PT:=T#200MS);
IF rtClearBelt[1].Q THEN
	iClearBeltStep:=88;//皮带清料触发
END_IF;

CASE iClearBeltStep OF
///////////////////////////////////////////////////////////凸轮耦合/////////////////////////////////////////////////////
88://有关气缸动作
	arrCyCtrl[CYNo.NGRevBeltTension].Cmd.bON:=TRUE;
	arrCyCtrl[CYNo.NGRevBeltUpDown].Cmd.bON:=TRUE;
	arrCyCtrl[CYNo.DustRevBeltUpDown].Cmd.bON:=TRUE;
	IF	arrCyCtrl[CyNo.NGRevBeltUpDown].Status.ONState AND arrCyCtrl[CYNo.DustRevBeltUpDown].Status.ONState THEN
		iClearBeltStep:=90;//		
	END_IF
	
90://凸轮/张力解耦
	bMethodTenBufferDisEnable:=TRUE;
	bMethodCamDisEnable:=TRUE;
	iClearBeltStep:=100;//	
	
100://判断是否解耦完成
	IF NOT bMethodTenBufferDisEnable AND NOT bMethodCamDisEnable THEN
		iClearBeltStep:=110;
	END_IF
110://主轴清0
	IF arrAxisCtrl[VirAxisNo.VirMain].Status.fModuloActPos<>0 THEN
		arrAxisCtrl[VirAxisNo.VirMain].Cmd.fSetPos:=arrAxisCtrl[VirAxisNo.VirMain].Status.fActPos-arrAxisCtrl[VirAxisNo.VirMain].Status.fModuloActPos+360;
		arrAxisCtrl[VirAxisNo.VirMain].Cmd.bSetPos:=TRUE;
	END_IF
	iClearBeltStep:=120;
120://皮带虚轴耦合
	IF NOT stVirBeltCam.bInSync THEN
		stVirBeltCam.bCamInExecute:=TRUE;
	ELSE
		iClearBeltStep:=130;
	END_IF	
130://皮带齿合
	IF NOT stCuterBeltGear.bInGear THEN
		stCuterBeltGear.bEnable:=TRUE;
	END_IF	
	IF NOT stNGReverseBeltGear.bInGear THEN
		stNGReverseBeltGear.bEnable:=TRUE;
	END_IF		
	IF NOT stDedustBeltGear.bInGear THEN
		stDedustBeltGear.bEnable:=TRUE;
	END_IF
	IF NOT stDedustReverseBeltGear.bInGear THEN
		stDedustReverseBeltGear.bEnable:=TRUE;
	END_IF

	IF NOT stSubBelt1Gear.bInGear THEN
		stSubBelt1Gear.bEnable:=TRUE;
	END_IF

	IF NOT stSubBelt2Gear.bInGear THEN
		bSubBelt2fratio:=TRUE;
		stSubBelt2Gear.bEnable:=TRUE;
	END_IF	
	
	IF NOT stSubBelt3Gear.bInGear THEN
		bSubBelt3fratio:=TRUE;
		stSubBelt3Gear.bEnable:=TRUE;
	END_IF		

	IF stCuterBeltGear.bInGear AND stNGReverseBeltGear.bInGear AND stDedustBeltGear.bInGear AND stDedustReverseBeltGear.bInGear AND 
	     stSubBelt1Gear.bInGear AND  stSubBelt2Gear.bInGear AND  stSubBelt3Gear.bInGear THEN
    	iClearBeltStep:=140;		
	END_IF
140://主轴运动40个周期
	arrAxisCtrl[VirAxisNo.VirMain].Cmd.bDynamitcsParSel:=1;
	arrAxisCtrl[VirAxisNo.VirMain].Cmd.fPositon_of_Abs:=arrAxisCtrl[VirAxisNo.VirMain].Status.fActPos-arrAxisCtrl[VirAxisNo.VirMain].Status.fModuloActPos+40*360;
	arrAxisPar[VirAxisNo.VirMain].fVelocity_of_Abs:=PolePar.iMainVel*6;
	arrAxisCtrl[VirAxisNo.VirMain].Cmd.bMoveAbs:=TRUE;
	IF arrAxisCtrl[VirAxisNo.VirMain].Status.Moving THEN
		iClearBeltStep:=150;
	END_IF
150://判断主轴运动完成
	IF arrAxisCtrl[VirAxisNo.VirMain].Status.NoMoving AND NOT arrAxisCtrl[VirAxisNo.VirMain].Cmd.bMoveAbs THEN
		iClearBeltStep:=160;
	END_IF
160://清除皮带记忆
	MEMSET(ADR(BeltData),0,SIZEOF(BeltData));
	iClearBeltStep:=170;
170://
	SysPart.hmiClearBelt:=FALSE;
	iClearBeltStep:=666;

END_CASE
END_ACTION

ACTION Product:

//切刀计数
rtCount2(CLK:=arrAxisCtrl[VirAxisNo.VirMain].Status.fModuloActPos>=10 AND arrAxisCtrl[VirAxisNo.VirMain].Status.fModuloActPos<=100);
IF rtCount2.Q THEN
	Production.OutFlag1:=TRUE;//产能计数
END_IF

////////////////////////////////////////////////////////////////NG剔废////////// NG分类 //////////////////////////////////////////////////////
ProductPar.iModeEN.bNG1PushEN:=ProductPar.iModeEN.bNG2PushEN;
CASE iNGStep OF 
10://判断NG1&NG2是否动作 主轴静止或运行中
	IF (  NOT ProductPar.iModeEN.bEmptyRunEN AND NOT ProductPar.iModeEN.bSizeCCDEN AND BeltData[BeltNo.NGBox1+2].fPoleNGSizeNo<>30 ) THEN//BeltData[BeltNo.NGBox].iPanoramaNG<>1
		 iNGStep:=200;
	ELSIF  BeltData[BeltNo.NGBox1+2].fPoleNGSacnNo<>30   AND NOT ProductPar.iModeEN.bLineScanCCDEN  THEN //XianSaong_Up[2]<>30 OR XianSaong_Down[0]<>30  
		iNGStep:=300;
	ELSIF  BeltData[BeltNo.NGBox1+2].bYellowMark    OR  BeltData[BeltNo.NGBox1+2].bBlueMark  THEN//黄标
		iNGStep:=300;
	ELSE
		nInt[3]:=0;
		arrCyCtrl[EvNo.	NGPushInsideAir	].Cmd.bON:=FALSE;//踢NG料打开
		arrCyCtrl[EvNo.	NGPushInsideAir	].Cmd.bOFF:=TRUE;//踢NG料关闭		
		arrCyCtrl[EVNo.NGPushInsideVacuo].Cmd.bON:=TRUE;//踢NG料真空打开
		arrCyCtrl[EVNo.NGPushInsideVacuo].Cmd.bOFF:=FALSE;//踢NG料真空关闭		
		iNGStep:=666;
	END_IF

200:
	IF  NOT ProductPar.iModeEN.bEmptyRunEN   THEN//AND NOT  ProductPar.iModeEN.bP2PartEN
			IF REAL_TO_INT(BeltData[BeltNo.NGBox1+2].fPoleNGSizeNo)=1 THEN
				Production.NGFlag[49]:=TRUE;//尺寸总不良
				Production.NGFlag[1]:=TRUE;//极片长度不良
			ELSIF REAL_TO_INT(BeltData[BeltNo.NGBox1+2].fPoleNGSizeNo)=2 THEN
				Production.NGFlag[49]:=TRUE;//尺寸总不良
				Production.NGFlag[2]:=TRUE;//极片CIL宽度不良
			ELSIF REAL_TO_INT(BeltData[BeltNo.NGBox1+2].fPoleNGSizeNo)=3 THEN
				Production.NGFlag[49]:=TRUE;//尺寸总不良
				Production.NGFlag[3]:=TRUE;//极片宽度不良标志位
			ELSIF REAL_TO_INT(BeltData[BeltNo.NGBox1+2].fPoleNGSizeNo)=4 THEN
				Production.NGFlag[49]:=TRUE;//尺寸总不良
				Production.NGFlag[4]:=TRUE;//极耳宽度不良
			ELSIF REAL_TO_INT(BeltData[BeltNo.NGBox1+2].fPoleNGSizeNo)=5 THEN
				Production.NGFlag[49]:=TRUE;//尺寸总不良
				Production.NGFlag[5]:=TRUE;//极耳高度不良
			ELSIF REAL_TO_INT(BeltData[BeltNo.NGBox1+2].fPoleNGSizeNo)=6 THEN
				Production.NGFlag[49]:=TRUE;//尺寸总不良
				Production.NGFlag[6]:=TRUE;//极耳侧边距不良
			ELSIF REAL_TO_INT(BeltData[BeltNo.NGBox1+2].fPoleNGSizeNo)=7 THEN
				Production.NGFlag[49]:=TRUE;//尺寸总不良
				Production.NGFlag[7]:=TRUE;//极耳面积不良
			ELSIF REAL_TO_INT(BeltData[BeltNo.NGBox1+2].fPoleNGSizeNo)=8 THEN
				Production.NGFlag[49]:=TRUE;//尺寸总不良
				Production.NGFlag[8]:=TRUE;//圆角深度不良
			ELSIF REAL_TO_INT(BeltData[BeltNo.NGBox1+2].fPoleNGSizeNo)=9 THEN
				Production.NGFlag[49]:=TRUE;//尺寸总不良
				Production.NGFlag[9]:=TRUE;//极耳边缘角度不良
			ELSIF REAL_TO_INT(BeltData[BeltNo.NGBox1+2].fPoleNGSizeNo)=10 THEN
				Production.NGFlag[49]:=TRUE;//尺寸总不良
				Production.NGFlag[10]:=TRUE;//圆角宽度不良
			ELSIF REAL_TO_INT(BeltData[BeltNo.NGBox1+2].fPoleNGSizeNo)=11 THEN
				Production.NGFlag[49]:=TRUE;//尺寸总不良
				Production.NGFlag[11]:=TRUE;//圆角轮廓不良	
			ELSIF REAL_TO_INT(BeltData[BeltNo.NGBox1+2].fPoleNGSizeNo)=12 THEN
				Production.NGFlag[49]:=TRUE;//尺寸总不良
				Production.NGFlag[12]:=TRUE;//圆角面积不良		
			ELSIF REAL_TO_INT(BeltData[BeltNo.NGBox1+2].fPoleNGSizeNo)=13 THEN
				Production.NGFlag[49]:=TRUE;//尺寸总不良
				Production.NGFlag[13]:=TRUE;//圆角余料不良		
			ELSIF (BeltData[BeltNo.NGBox1+2].fPoleNGSizeNo<>1 AND BeltData[BeltNo.NGBox1+2].fPoleNGSizeNo<>2 AND BeltData[BeltNo.NGBox1+2].fPoleNGSizeNo<>3
				AND BeltData[BeltNo.NGBox1+2].fPoleNGSizeNo<>4 AND BeltData[BeltNo.NGBox1+2].fPoleNGSizeNo<>5 AND BeltData[BeltNo.NGBox1+2].fPoleNGSizeNo<>6
				 AND BeltData[BeltNo.NGBox1+2].fPoleNGSizeNo<>7  AND BeltData[BeltNo.NGBox1+2].fPoleNGSizeNo<>8  AND BeltData[BeltNo.NGBox1+2].fPoleNGSizeNo<>9
				 AND BeltData[BeltNo.NGBox1+2].fPoleNGSizeNo<>11  AND BeltData[BeltNo.NGBox1+2].fPoleNGSizeNo<>12  AND BeltData[BeltNo.NGBox1+2].fPoleNGSizeNo<>13
				) OR  BeltData[BeltNo.NGBox1+2].fPoleNGSizeNo=33  THEN  //尺寸检测其他不良 ,,,CCD超时
				Production.NGFlag[49]:=TRUE;//尺寸检测其他不良 ,,,CCD超时
				Production.NGFlag[14]:=TRUE;
			END_IF
	END_IF
		FOR i:=1 TO 20 DO
			IF i<20 THEN
				XianSaong[21-i]:=XianSaong[20-i];
				XianSaong1[21-i]:=XianSaong1[20-i];
			ELSE
				XianSaong[1]:=BeltData[BeltNo.NGBox1].iPanoramaNG;
				XianSaong1[1]:=REAL_TO_INT(BeltData[BeltNo.NGBox1].fPoleNGSizeNo);
			END_IF
		END_FOR
		iNGStep:=400;
300:
	 IF NOT ProductPar.iModeEN.bEmptyRunEN  THEN//AND NOT  ProductPar.iModeEN.bP2PartEN
			IF BeltData[BeltNo.NGBox1+2].fPoleNGSacnNo=1 THEN
				Production.NGFlag[48]:=TRUE;//线扫总不良
				Production.NGFlag[21]:=TRUE;//抓边失败
			ELSIF BeltData[BeltNo.NGBox1+2].fPoleNGSacnNo=2 THEN
				Production.NGFlag[48]:=TRUE;//线扫总不良
				Production.NGFlag[22]:=TRUE;//直边不良标志位
			ELSIF BeltData[BeltNo.NGBox1+2].fPoleNGSacnNo=3 THEN
				Production.NGFlag[48]:=TRUE;//线扫总不良
				Production.NGFlag[23]:=TRUE;//极片缺失
			ELSIF BeltData[BeltNo.NGBox1+2].fPoleNGSacnNo=4 THEN
				Production.NGFlag[48]:=TRUE;//线扫总不良
				Production.NGFlag[24]:=TRUE;//接带
			ELSIF BeltData[BeltNo.NGBox1+2].fPoleNGSacnNo=5 THEN
				Production.NGFlag[48]:=TRUE;//线扫总不良
				Production.NGFlag[25]:=TRUE;//线扫黄标
			ELSIF BeltData[BeltNo.NGBox1+2].fPoleNGSacnNo=6 THEN
				Production.NGFlag[48]:=TRUE;//线扫总不良
				Production.NGFlag[26]:=TRUE;//漏金属
			ELSIF BeltData[BeltNo.NGBox1+2].fPoleNGSacnNo=7 THEN
				Production.NGFlag[48]:=TRUE;//线扫总不良
				Production.NGFlag[27]:=TRUE;//气泡
			ELSIF BeltData[BeltNo.NGBox1+2].fPoleNGSacnNo=8 THEN
				Production.NGFlag[48]:=TRUE;//线扫总不良
				Production.NGFlag[28]:=TRUE;//暗条痕
			ELSIF BeltData[BeltNo.NGBox1+2].fPoleNGSacnNo=9 THEN
				Production.NGFlag[48]:=TRUE;//线扫总不良
				Production.NGFlag[29]:=TRUE;//亮条痕
			ELSIF BeltData[BeltNo.NGBox1+2].fPoleNGSacnNo=10 THEN
				Production.NGFlag[48]:=TRUE;//线扫总不良
				Production.NGFlag[30]:=TRUE;//破损
			ELSIF BeltData[BeltNo.NGBox1+2].fPoleNGSacnNo=11 THEN
				Production.NGFlag[48]:=TRUE;//线扫总不良
				Production.NGFlag[31]:=TRUE;//碎屑
			ELSIF BeltData[BeltNo.NGBox1+2].fPoleNGSacnNo=12 THEN
				Production.NGFlag[48]:=TRUE;//线扫总不良
				Production.NGFlag[33]:=TRUE;//脱碳
			ELSIF BeltData[BeltNo.NGBox1+2].fPoleNGSacnNo=29 THEN
				Production.NGFlag[48]:=TRUE;//线扫总不良
				Production.NGFlag[34]:=TRUE;//其他
			ELSIF BeltData[BeltNo.NGBox1+2].fPoleNGSacnNo=33 THEN
				Production.NGFlag[48]:=TRUE;//线扫总不良
				Production.NGFlag[32]:=TRUE;//通讯超时
(*			ELSIF BeltData[BeltNo.NGBox1+2].bYellowMark  THEN
				//Production.NGFlag[48]:=TRUE;//线扫总不良
				Production.NGFlag[33]:=TRUE;//感应器黄标*)
			END_IF
	END_IF
		iNGStep:=400;
400:
	arrCyCtrl[EvNo.	NGPushInsideAir	].Cmd.bON:=TRUE;//踢NG料破真空打开
	arrCyCtrl[EvNo.	NGPushInsideAir	].Cmd.bOFF:=FALSE;//踢NG料破真空关闭
	arrCyCtrl[EVNo.NGPushInsideVacuo].Cmd.bON:=FALSE;//踢NG料真空打开
	arrCyCtrl[EVNo.NGPushInsideVacuo].Cmd.bOFF:=TRUE;//踢NG料真空关闭
	BeltData[BeltNo.NGBox1+2].bHavePole:=FALSE;	
	BeltData[BeltNo.NGBox1+2].stPoleNo:='';
	nInt[3]:=1;		
	//BeltData[BeltNo.NGBox1].bHavePole:=FALSE;
	FOR i:=1 TO 50 DO//NG类型标志位复位
		Production.NGFlag[i]:=FALSE;
    	END_FOR
	iNGStep:=666;
END_CASE

IF iNGStep=300 THEN
	IF BeltData[BeltNo.NGBox1+1].bBlueMark OR BeltData[BeltNo.NGBox1+2].bBlueMark OR BeltData[BeltNo.NGBox1+3].bBlueMark THEN
		iNGState:=1;//接带踢废
	ELSIF BeltData[BeltNo.NGBox1+2].bYellowMark THEN
		IF BeltData[BeltNo.NGBox1+1].bYellowMark THEN
			iNGState:=2;//黄标跳切踢废
		ELSIF NOT BeltData[BeltNo.NGBox1+3].bYellowMark THEN
			iNGState:=3;//黄标单张踢废
		END_IF
	ELSIF BeltData[BeltNo.NGBox1+2].fPoleNGSacnNo=4 THEN
		iNGState:=4;//线扫接带
	ELSIF BeltData[BeltNo.NGBox1+2].fPoleNGSacnNo=5 THEN
		iNGState:=5;//线扫黄标
	END_IF
END_IF

aFB_ProductionDataLocal(
	NowTimeData:=System.StTime, (*当前系统时间*)
	OutFlag1:=Production.OutFlag1, (*产量计数标志1*)
	OutFlag2:=Production.OutFlag2, (*产量计数标志1*)
	NGFlag:=Production.NGFlag ,(*NG1计数标志*)(*扫码NG*)
	RunFlag:=stSysState.iMode=1,(*运行标志*)
	WaitFlag:=stSysState.iMode<>1 AND NOT stSysState.Alarming ,(*待料标志*)
	AlarmFlag:=stSysState.Alarming, (*故障标志*)
	DelDataAMBtn:= Production.HMI_DelDataAMBtn,(*白班数据清除按钮*)//HMI_DayCountZero
	DelDataPMBtn:= Production.HMI_DelDataPMBtn,(*夜班数据清除按钮*)//HMI_NightCountZero
	NowOutTotal=>Production.HMI_TotalCount ,(*当前班次加工总数*)
	NowRate=> Production.HMI_Qualified,(*当前班次良率*)
	NGClearAMBtn:=Production.HMI_NGClearAMBtn,//白班NG类型计数清零
	NGClearPMBtn:=Production.HMI_NGClearPMBtn,//夜班NG类型计数清零
	NowDay:= Production.SaveNowDay,(*数据移位时所保存当前日*)
	NowMonth:=Production.SaveNowMonth ,(*数据移位时所保存当前月*)
	DayHistory:= Production.DayReadDayHistory, (*历史日*)
	MonthHistory:= Production.DayReadMonthHistory,(*历史月*)
	TodayTotal:=Production.HMI_TodayTotal ,(*当天24H生产总数*)
	TodayOK:=Production.HMI_TodayOK , (*当天24H生产OK总数*)
	TodayNG:=Production.HMI_TodayNG , (*当天24H生产NG总数*)
	TodayTotal_AM:= Production.DayCountTotal,(*当天白班生产总数*)
	TodayTotal_PM:=Production.NightCountTotal,(*当天夜班生产总数*)
	TodayRate_AM:= Production.HMI_DayQualified,(*当天白班良率*)
	TodayRate_PM:=Production.HMI_NightQualified ,(*当天夜班良率*)
	OEE=> Production.HMI_OEE,//设备稼动率/稼动率
	TodayOK_AM:=Production.HMI_DayOkCount ,(*当天白班生产OK总数*)
	TodayOK_PM:= Production.HMI_NightOkCount,(*当天夜班生产OK总数*)
	TodayNG_AM:=Production.HMI_DayNgCount ,(*当天白班生产NG总数*)
	TodayNG_PM:=Production.HMI_NightNgCount , (*当天夜班生产NG总数*)
	TodayHour_AM:= Production.HourTimeDayCount,(*当天白班每小时产量ARRAY[8..19 ]*)
	TodayHour_PM:=Production.HourTimeNightCount ,(*当天夜班每小时产量ARRAY[0..23]*)
	TodayNGClass_AM:=Production.NgPerHourDayCount , (*当天白班各类NG数量ARRAY[1..30 ]*)
	TodayNGClass_PM:= Production.NgPerHourNightCount,(*当天夜班各类NG数量ARRAY[1..30 ]*)
	TodayRun_AM:= Production.DayRunTimeTotal,(*当天白班总运行时间合计/分*)
	TodayRun_PM:= Production.NightRunTimeTotal,(*当天夜班总运行时间合计/分*)
	TodayWait_AM:=Production.DayWaitTimeTotal , (*当天白班总待料时间合计/分*)
	TodayWait_PM:=Production.NightWaitTimeTotal , (*当天夜班总待料时间合计/分*)
	TodayAlarm_AM:=Production.DayAlarmTimeTotal ,(*当天白班总报警时间合计/分*)
	TodayAlarm_PM:=Production.NightAlarmTimeTotal, (*当天夜班总报警时间合计/分*)
	
	TodayRun_AMH:=Production.DayRunTime_min,(*当天白班每小时运行时间合计/分*)
	TodayRun_PMH:=Production.NightRunTime_min,(*当天夜班每小时运行时间合计/分*)
	TodayWait_AMH:=Production.DayWaitTime_min,(*当天白班每小时待料时间合计/分*)
	TodayWait_PMH:=Production.NightWaitTime_min,(*当天夜班每小时待料时间合计/分*)
	TodayAlarm_AMH:=Production.DayAlmTime_min,(*当天白班每小时报警时间合计/分*)
	TodayAlarm_PMH:=Production.NightAlmTime_min,(*当天夜班每小时报警时间合计/分*)
	
	HistoryRun_AMH:=Production.HisDayRunTime_min,(*历史每天白班每小时运行时间合计ARRAY[1..7 ]*)
	HistoryRun_PMH:=Production.HisNightRunTime_min,(*历史每天夜班每小时运行时间合计ARRAY[1..7 ]*)
	HistoryWait_AMH:=Production.HisDayWaitTime_min,(*历史每天白班每小时待料时间合计ARRAY[1..7 ]*)
	HistoryWait_PMH:=Production.HisNightWaitTime_min,(*历史每天夜班每小时待料时间合计ARRAY[1..7 ]*)
	HistoryAlarm_AMH:=Production.HisDayAlmTime_min,(*历史每天白班每小时报警时间合计ARRAY[1..7 ]*)
	HistoryAlarm_PMH:=Production.HisNightAlmTime_min,(*历史每天夜班每小时报警时间合计ARRAY[1..7 ]*)
	
	RunCnt_AM:=Production.nDayRunTimeCnt , (*白班运行时间计数*)
	RunCnt_PM:=Production.nNightRunTimeCnt ,(*夜班运行时间计数*)
	WaitCnt_AM:= Production.nDayWaitTimeCnt, (*白班待料时间计数*)
	WaitCnt_PM:=Production.nNightWaitTimeCnt ,(*夜班待料时间计数*)
	AlarmCnt_AM:=Production.nDayAlarmTimeCnt , (*白班报警时间计数*)
	AlarmCnt_PM:= Production.nNightAlarmTimeCnt,(*夜班报警时间计数*)
	
	HistoryTotal:=Production.HMI_HistoryTotal ,(*历史每天24H生产总数ARRAY[1..7 ]*)
	HistoryOK:=Production.HMI_HistoryOK ,(*历史每天24H生产OK总数ARRAY[1..7 ]*)
	HistoryNG:=Production.HMI_HistoryNG , (*历史每天24H生产NG总数ARRAY[1..7 ]*)
	HistoryTotal_AM:=Production.DayCountTotalHistory ,(*历史每天白班生产总数ARRAY[1..7 ]*)
	HistoryTotal_PM:=Production.NightCountTotalHistory ,(*历史每天夜班生产总数ARRAY[1..7 ]*)
	HistoryRate_AM:=Production.HMI_DayQualifiedHistory , (*历史每天白班良率ARRAY[1..7 ]*)
	HistoryRate_PM:=Production.HMI_NightQualifiedHistory,(*历史每天夜班良率ARRAY[1..7 ]*)
	HistoryOK_AM:=Production.HMI_DayOkCountHistory , (*历史每天白班生产OK总数ARRAY[1..7 ]*)
	HistoryOK_PM:=Production.HMI_NightOkCountHistory , (*历史每天夜班生产OK总数ARRAY[1..7 ]*)
	HistoryNG_AM:=Production.HMI_DayNgCountHistory ,(*历史每天白班生产NG总数ARRAY[1..7 ]*)
	HistoryNG_PM:= Production.HMI_NightNgCountHistory,(*历史每天夜班生产NG总数ARRAY[1..7 ]*)
	HistoryHour_AM:=Production.HourTimeDayCountHistory ,(*历史每天白班每小时产量ARRAY[1..7,8..19 ]*)
	HistoryHour_PM:=Production.HourTimeNightCountHistory ,(*历史每天夜班每小时产量ARRAY[1..7,0..23]*)
	HistoryNGClass_AM:= Production.NgPerHourDayCountHistory,(*历史每天白班各类NG数量ARRAY[1..7,1..30 ]*)
	HistoryNGClass_PM:= Production.NgPerHourNightCountHistory,(*历史每天夜班各类NG数量ARRAY[1..7,1..30 ]*)
	HistoryRun_AM:=Production.DayRunTimeTotalHistory , (*历史每天白班总运行时间合计ARRAY[1..7 ]*)
	HistoryRun_PM:= Production.NightRunTimeTotalHistory, (*历史每天夜班总运行时间合计ARRAY[1..7 ]*)
	HistoryWait_AM:= Production.DayWaitTimeTotalHistory,(*历史每天白班总待料时间合计ARRAY[1..7 ]*)
	HistoryWait_PM:= Production.NightWaitTimeTotalHistory, (*历史每天夜班总待料时间合计ARRAY[1..7 ]*)
	HistoryAlarm_AM:= Production.DayAlarmTimeTotalHistory,(*历史每天白班总报警时间合计ARRAY[1..7 ]*)
	HistoryAlarm_PM:= Production.NightAlarmTimeTotalHistory,(*历史每天夜班总报警时间合计ARRAY[1..7 ]*)

	TodayNgHour_Day:=Production.HMINgClassCount_Day,(*白班每种NG类型每小时统计 ,,,NG类型，小时*)
	TodayNgHour_Night:=Production.HMINgClassCount_Night,(*夜班每种NG类型每小时统计 ,,,NG类型，小时*)
	HisTodayNgHour_Day:=Production.HisHMINgClassCount_Day,//l历史白班每小时NG类型统计,,
	HisTodayNgHour_Night:=Production.HisHMINgClassCount_Night,//历史夜班每小时NG类型统计,,
		
	TodayNGQualified:=Production.HMI_TodayNGQualified,//当天白班各种NG类型NG率
	NightNGQualified:=Production.HMI_NightNGQualified,//当天夜班各种NG类型NG率	
	HisTodayNGQualified:=Production.HMI_HisTodayNGQualified,//历史白班各种NG类型NG率
	HisNightNGQualified:=Production.HMI_HisNightNGQualified,//历史夜班各种NG类型NG率
	
	);
END_ACTION

END_FUNCTION_BLOCK

(* stored: Version 1.1.0.1, ProductVersion 3.1.4024.12
   POU FB_UserMain: Id {f8fe3f95-1222-48ed-9589-1065369e5491}, SpecialFunc None
   Folder F05Auto: Id {210754a1-66db-40ea-b245-f03d86e51ef2}
   Action Alarm: Id {0dd32a61-1957-4014-a4d5-7c49efa314d3}
   Action F00Home: Id {9fe7157e-5263-4fea-8306-1300724fdeaa}
   Action F01MotionManual: Id {899cecb5-0461-4078-9f42-e4d36a44648f}
   Action F02CylinderManual: Id {051cf36c-698c-410d-b744-a8fb64c5fc87}
   Action F03FunctionTen: Id {0e98ed10-037e-4015-85d2-f5f1da96dc98}
   Action F04FunctionCam: Id {d40e8d1d-579a-4abd-8f8c-68db7e4f1147}
   Action F0500MainAuto: Id {4bd03534-9f1c-4caf-84b4-910a0cc987a6}
   Action F0501MainAuto1: Id {9418259e-13d2-47ae-a72e-4ee7e4cb4033}
   Action F0502MainAuto2: Id {2dfdd34e-1280-4a35-9637-7024e7eba164}
   Action F0503MainAuto3: Id {03bd2d44-14eb-4799-82e4-91e79713d961}
   Action F0504MainAuto4: Id {3d3a323e-c4a0-4052-8891-4bef7111eefe}
   Action F0505MainAuto5: Id {b39cfad9-81c8-4946-bcd6-65c257ac9bf0}
   Action F0506MainAuto6: Id {ced1a7f7-55cc-47a7-961f-0d671a532305}
   Action F0511CCDAuto: Id {f14efd26-61eb-4417-b8c9-391a17c82217}
   Action F0512CarryAuto: Id {67df423c-8635-4b02-afc7-784b57f3064b}
   Action F0599AutoAux: Id {fd0c7923-717c-41e5-9f37-2adcbf7f5731}
   Action F05Rectifydev: Id {6d1368d9-9736-4802-a465-2be8ef0291f5}
   Action F07Condition: Id {051551c2-babe-4355-b6ce-48d75c0b401e}
   Action F09INIT: Id {3694dc3b-44dc-46c1-b718-edddb24dbb6f}
   Action F10GearCall: Id {21106b04-cadb-4aee-a9ed-00cdd1d15078}
   Action F11CamCall: Id {0d2bf613-8ddc-4699-a88f-83f349d84534}
   Action F12TensionCall: Id {773d1077-f8f5-4c07-aa80-533245b96411}
   Action F13ClearBelt: Id {d22918f8-1cb8-494b-a07f-103510ff5d58}
   Action Product: Id {50221cb1-87b1-443c-9509-e84508d0df40} *)
